FUNCTION_BLOCK SoftPWM (* PWM output *)
  (* Standard: 61499-2 *)
  (* Version 1.0, 2026-04-18, Thomas Mayr *)
  PACKAGE iec61499::events;
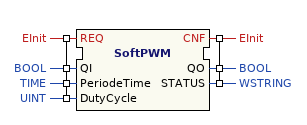
  EVENT_INPUT
    REQ : EInit WITH PeriodeTime, DutyCycle, QI; (* Service Initialization *)
  END_EVENT
  EVENT_OUTPUT
    CNF : EInit WITH QO, STATUS; (* Initialization Confirm *)
  END_EVENT
  VAR_INPUT
    QI : BOOL; (* Event Input Qualifier *)
    PeriodeTime : TIME; (* Time of each Periode *)
    DutyCycle : UINT; (* Duty Cycle in Percent *)
  END_VAR
  VAR_OUTPUT
    QO : BOOL; (* Event Output Qualifier *)
    STATUS : WSTRING; (* Service Status *)
  END_VAR
END_FUNCTION_BLOCK
